(* PLC project MotionTest, Beckhoff Automation GmbH TwinCAT PLC Control 3.5.13.21 *)
(* stored: creationDateTime 2025-04-03T14:51:11.685745, modificationDateTime 2025-04-03T14:51:11.685745 *)

{attribute 'qualified_only'}
{attribute 'strict'}
TYPE MotorState :
(
    NONE        ,
    STARTING_MOTOR,
    MOVE_TO_A     ,
    MOVE_TO_B     ,
    STOPPING_MOTOR
);
END_TYPE
